// TwinCAT 3 PLC project TF6620_S7CommunicationSamplePlc
// ProgramVersion: 3.1.4023.0
// libraries:
//   Tc2_Standard, * (Beckhoff Automation GmbH)
//   Tc2_System, * (Beckhoff Automation GmbH)
//   Tc3_Module, * (Beckhoff Automation GmbH)
//   Tc3_S7Comm, * (Beckhoff Automation GmbH)
// project tree:
//   DUTs/ ST_S7_Incoming.TcDUT, ST_S7_Incoming_Cyclic.TcDUT (not stored), ST_S7_Info.TcDUT (not stored), ST_S7_RequestHandling.TcDUT (not stored)
//   / PlcTask.TcTTO
//   POUs/ MAIN.TcPOU, MAIN2.TcPOU
// real-time tasks:
//   TASK PlcTask: cycle T#10ms, priority 20, ADS port 350
// I/O:
//   DEVICE Device 1 (RT-Ethernet Adapter)
// variable links:
//   TF6620_S7CommunicationSamplePlc/TF6620_S7CommunicationSamplePlc Instance <-> Device 1 (RT-Ethernet Adapter)/Device 1 (RT-Ethernet Adapter)_Obj1 (TCP/UDP RT)/Object1 (S7 Connector)
//     PlcTask Inputs/MAIN.stS7Info.bS7Error <-> Status/Error
//     PlcTask Inputs/MAIN.stS7Info.eS7CommState <-> Status/State
//   TF6620_S7CommunicationSamplePlc/TF6620_S7CommunicationSamplePlc Instance <-> Device 1 (RT-Ethernet Adapter)/Device 1 (RT-Ethernet Adapter)_Obj1 (TCP/UDP RT)/Object1 (S7 Connector)/Object1 (S7 Single Request)
//     PlcTask Inputs/MAIN.stS7Incoming.b{1..4} <-> ReadFromS7/b{1..4}  (4 links)
//     PlcTask Inputs/MAIN.stS7Incoming.by1 <-> ReadFromS7/by1
//     PlcTask Inputs/MAIN.stS7Incoming.i1 <-> ReadFromS7/i1
//     PlcTask Inputs/MAIN.stS7Incoming.r1 <-> ReadFromS7/r1
//     PlcTask Inputs/MAIN.stS7Incoming.r2 <-> ReadFromS7/r2
//     PlcTask Inputs/MAIN.stS7Incoming.w1 <-> ReadFromS7/w1
//     PlcTask Inputs/MAIN.stS7Info.nError <-> Status/Error
//     PlcTask Inputs/MAIN.stS7RequestHandling.byReceiveCounter <-> Status/ReceiveCounter
//     PlcTask Outputs/MAIN.bWriteEnable <-> Control/WriteToS7Enable
//     PlcTask Outputs/MAIN.i1write <-> WriteToS7/i1
//     PlcTask Outputs/MAIN.stS7RequestHandling.bySendRequest <-> Control/SendRequest
//   TF6620_S7CommunicationSamplePlc/TF6620_S7CommunicationSamplePlc Instance <-> Device 1 (RT-Ethernet Adapter)/Device 1 (RT-Ethernet Adapter)_Obj1 (TCP/UDP RT)/Object1 (S7 Connector)/Object2 (S7 Cycle Request)
//     PlcTask Inputs/MAIN.stS7IncomingCyclic.b{1..4} <-> ReadFromS7/b{1..4}  (4 links)
//     PlcTask Inputs/MAIN.stS7IncomingCyclic.by1 <-> ReadFromS7/by1
//     PlcTask Inputs/MAIN.stS7IncomingCyclic.i1 <-> ReadFromS7/i1
//     PlcTask Inputs/MAIN.stS7IncomingCyclic.r1 <-> ReadFromS7/r1
//     PlcTask Inputs/MAIN.stS7IncomingCyclic.r2 <-> ReadFromS7/r2
//     PlcTask Inputs/MAIN.stS7IncomingCyclic.w1 <-> ReadFromS7/w1

CONFIGURATION TF6620_S7CommunicationSamplePlc
    RESOURCE PLC ON TwinCAT3
        TASK PlcTask(INTERVAL := T#10ms, PRIORITY := 20);
        PROGRAM MAIN WITH PlcTask : MAIN;
        PROGRAM MAIN2 WITH PlcTask : MAIN2;
    END_RESOURCE
END_CONFIGURATION

// ---- DUTs/ST_S7_Incoming.TcDUT
TYPE ST_S7_Incoming :
STRUCT
	by1 AT%I* 	: BYTE;
	b1 AT%I* 	: BOOL;
	b2 AT%I* 	: BOOL;
	b3 AT%I* 	: BOOL;
	b4 AT%I* 	: BOOL;
	w1 AT%I*	: DWORD;
	r1 AT%I*	: REAL;
	r2 AT%I*	: REAL;
	i1 AT%I*	: INT;	
END_STRUCT
END_TYPE

// ---- POUs/MAIN.TcPOU
PROGRAM MAIN
VAR
	bStartReadRequest 	: BOOL;	
	bStartWriteRequest	: BOOL;
	
	stS7Info			: ST_S7_Info;
	stS7RequestHandling	: ST_S7_RequestHandling;

	(* Read variables *)
	bReadRequestDone	: BOOL;
	stS7Incoming		: ST_S7_Incoming;
	stS7IncomingCyclic	: ST_S7_Incoming_Cyclic;
	
	(* Write variables *)
	bWriteEnable AT%Q*	: BOOL;
	bWriteRequestDone	: BOOL;
	i1write AT%Q*		: INT := 42;
	
	(* State machine variables *)
	nState				: UINT;
	nStateWrite			: UINT;
	
END_VAR

CASE nState OF 
	0: 
		IF bStartReadRequest THEN
			bStartReadRequest := FALSE;
			bReadRequestDone := FALSE;
			nState := nState + 1;
		END_IF

	1:
		stS7RequestHandling.bySendRequest := stS7RequestHandling.byReceiveCounter + 1;
		nState := nState + 1;
		
	2: 
		IF stS7RequestHandling.byReceiveCounter = stS7RequestHandling.bySendRequest THEN
			nState := nState + 1;
		END_IF	
		
	3: 
		bReadRequestDone := TRUE;
		nState := 0;
	
END_CASE

CASE nStateWrite OF
	0:
		IF bStartWriteRequest THEN
			bStartWriteRequest := FALSE;
			bWriteEnable := TRUE;
			nStateWrite := nStateWrite + 1;
		END_IF

	1:
		stS7RequestHandling.bySendRequest := stS7RequestHandling.byReceiveCounter + 1;
		nStateWrite := nStateWrite + 1;
		
	2: 
		IF stS7RequestHandling.byReceiveCounter = stS7RequestHandling.bySendRequest THEN
			bWriteEnable := FALSE;
			nStateWrite := nStateWrite + 1;
		END_IF	
	
	3: 
		bWriteRequestDone := TRUE;
		nStateWrite := 0;
		
END_CASE

END_PROGRAM

// ---- POUs/MAIN2.TcPOU
PROGRAM MAIN2
VAR
	bInitDone:	BOOL:=FALSE;
	
	fbConnection: FB_S7CommConnection(16#01010050);
	
	fbRequestRead   : FB_S7CommSingleRequest;
	fbRequestWrite  : FB_S7CommSingleRequest;
	fbRequestCyclic : FB_S7CommCyclicRequest;
	
	data_byte			: BYTE;
	data_dword			: DWORD;
	data_byte_cyclic	: BYTE;
	data_dword_cyclic	: DWORD;
	data_int_cyclic		: INT;
	
	data_counter: WORD;
	data_el1008: BYTE;
	data_el2008: BYTE;
	
	ipaddr:		IPADDR;
	hr:			HRESULT;
	bRead: BOOL := FALSE;
	bWrite: BOOL := FALSE;
	bReset:	BOOL := FALSE;
	bConnect:	BOOL := FALSE;
	connectionError:	STRING;	
	requestError:	STRING;

	a : S7COMM_CONNECT_STATE;
	nState:	UINT := 0;
END_VAR

IF NOT bInitDone THEN

	// Read
	fbRequestRead.AddReadVar(ADR(data_byte),  SIZEOF(data_byte),  0 * 8, S7COMM_DATAAREA_DATA_BLOCKS, 1);
	fbRequestRead.AddReadVar(ADR(data_dword), SIZEOF(data_dword), 2 * 8, S7COMM_DATAAREA_DATA_BLOCKS, 1);
	
	// write
	// fbRequestWrite.AddWriteVar(ADR(data_el2008), SIZEOF(data_el2008), 38 * 8, S7COMM_DATAAREA_OUTPUT, 0);
	
	// read cyclic
	fbRequestCyclic.AddReadVar(ADR(data_byte_cyclic),  SIZEOF(data_byte_cyclic),  0 * 8, S7COMM_DATAAREA_DATA_BLOCKS, 1);
	fbRequestCyclic.AddReadVar(ADR(data_dword_cyclic), SIZEOF(data_dword_cyclic), 2 * 8, S7COMM_DATAAREA_DATA_BLOCKS, 1);
	fbRequestCyclic.AddReadVar(ADR(data_int_cyclic), SIZEOF(data_int_cyclic), 14 * 8, S7COMM_DATAAREA_DATA_BLOCKS, 1);
	
		// add to connection
	fbConnection.AddRequest(fbRequestRead);	
	fbConnection.AddRequest(fbRequestWrite);	
	fbConnection.AddRequest(fbRequestCyclic);
	
	fbConnection.bExecute := FALSE;
	fbRequestWrite.bExecute := FALSE;
	fbRequestRead.bExecute := FALSE;
	fbRequestCyclic.bExecute := FALSE;
	
	bInitDone := TRUE;
	nState := 1;
END_IF


CASE nState OF
	// IDLE
	0:;
	
	// CONNECT
	1:
	IF bConnect THEN
		fbConnection.sIpAddr := '10.3.32.101';
		fbConnection.eCpuType := S7COMM_CPUTYPE_S71500;
		fbConnection.nRack := 0;
		fbConnection.nSlot := 0;
		
		fbConnection.bExecute := TRUE;
		bConnect := FALSE;
		nState := 10;
	END_IF
	
	// WAIT FOR CONNECT
	10:
	IF NOT fbConnection.bBusy THEN
		IF fbConnection.bError THEN
			connectionError := fbConnection.sErrorTxt;
			nState := 1000;
		ELSE
			fbRequestCyclic.nCycleTimeMs := 1000;
			fbRequestCyclic.bExecute := TRUE;
			nState := 20;
		END_IF
	END_IF
	
	// RUNNING
	20:
	IF bRead THEN
		bRead := FALSE;
		fbRequestRead.bExecute := TRUE;
		nState := 30;
	END_IF
	
	IF bWrite THEN
		bWrite := FALSE;
		fbRequestWrite.bExecute := TRUE;
		nState := 40;
	END_IF
	
	IF fbRequestCyclic.bError THEN
		requestError := fbRequestCyclic.sErrorTxt;
		nState := 1000;
	END_IF
	
	30:
	IF NOT fbRequestRead.bBusy THEN
		IF fbRequestRead.bError THEN
			requestError := fbRequestRead.sErrorTxt;
			nState := 1000;
		ELSE
			fbRequestRead.bExecute := FALSE;
			nState := 20;
		END_IF
	END_IF
	
	40:
	IF NOT fbRequestWrite.bBusy THEN
		IF fbRequestWrite.bError THEN
			requestError := fbRequestWrite.sErrorTxt;
			nState := 1000;
		ELSE
			fbRequestWrite.bExecute := FALSE;
			nState := 20;
		END_IF
	END_IF
	
	// ERROR
	1000:
	IF bReset THEN
		nState := 2000;
	END_IF
	
	// RESET
	2000:
		fbConnection.bExecute := FALSE;
		fbRequestWrite.bExecute := FALSE;
		fbRequestRead.bExecute := FALSE;
		fbRequestCyclic.bExecute := FALSE;
		connectionError := '';
		requestError := '';
		nState := 1;
END_CASE

// fb calls
fbConnection();
fbRequestRead();
fbRequestWrite();
fbRequestCyclic();

END_PROGRAM
